// TIA Portal V15.1 export
// export: Created 2024-06-21T08:40:58.6119821Z, ExportSetting WithDefaults, DisplayName Totally Integrated Automation Portal, DisplayVersion V15.1 Update 5, DisplayName TIA Portal Openness, DisplayVersion V15.1 Update 5, DisplayName SINAMICS Startdrive Advanced, DisplayVersion V15.1, DisplayName G130, G150, S120, S150, SINAMICS MV, S210, DisplayVersion V15.1, DisplayName G110M, G120, G120C, G120D, G120P, DisplayVersion V15.1, DisplayName STEP 7 Professional, DisplayVersion V15.1 Update 5, DisplayName STEP 7 Safety, DisplayVersion V15.1, DisplayName WinCC Professional, DisplayVersion V15.1 Update 5, DisplayName SIMATIC Visualization Architect, DisplayVersion V15.1
FUNCTION_BLOCK "LDP/PNCouplerDiag"   // FB1901, FBD
TITLE = LDPCouplerDiag
{ S7_Optimized_Access := 'FALSE' }
AUTHOR : VCC
FAMILY : Communic
NAME : LDPDiag
VERSION : 0.1
// ================================================================================
// Function used to read the diagnostic information from a DP/DP coupler.
// ================================================================================
// stored: AutoNumber false, IsIECCheckEnabled false, SetENOAutomatically False, UDAEnableTagReadback false
   VAR_INPUT
      I_PNPNSendError { ExternalAccessible := 'False'; ExternalVisible := 'False'; ExternalWritable := 'False'} : Bool;   // Send Error
      I_PNPNSendSUBSOn { ExternalAccessible := 'False'; ExternalVisible := 'False'; ExternalWritable := 'False'} : Bool;   // SUBS ON
      I_PNPNDiagSend { ExternalAccessible := 'False'; ExternalVisible := 'False'; ExternalWritable := 'False'} : Byte;   // Diag
      I_PNPNRcvError { ExternalAccessible := 'False'; ExternalVisible := 'False'; ExternalWritable := 'False'} : Bool;   // Recv Error
      I_PNPNRcvSUBSOn { ExternalAccessible := 'False'; ExternalVisible := 'False'; ExternalWritable := 'False'} : Bool;   // SUBS ON
      I_PNPNRcvAckReq { ExternalAccessible := 'False'; ExternalVisible := 'False'; ExternalWritable := 'False'} : Bool;   // ACK REQ
      I_PNPNDiagRecv { ExternalAccessible := 'False'; ExternalVisible := 'False'; ExternalWritable := 'False'} : Byte;   // Diag
      I_AlarmResetPB { ExternalAccessible := 'False'; ExternalVisible := 'False'; ExternalWritable := 'False'} : Bool;   // Alarm reset pushbutton is activated
   END_VAR
   VAR_OUTPUT
      O_Alarm { ExternalAccessible := 'False'; ExternalVisible := 'False'; ExternalWritable := 'False'} : Bool;   // Alarm
      O_AlarmABCondition { ExternalAccessible := 'False'; ExternalVisible := 'False'; ExternalWritable := 'False'} : Bool;   // Alarms AB condition
      H_IAnim { ExternalAccessible := 'False'; ExternalVisible := 'False'; ExternalWritable := 'False'} : Word;   // Icon Animation
   END_VAR
   VAR DB_SPECIFIC
      H_Out : Struct   // HMI
         Anim : Word;   // HMI Animation of the object
         DBnr : Int;   // HMI Animation DB number
      END_STRUCT;
      Alarm { ExternalAccessible := 'False'; ExternalVisible := 'False'; ExternalWritable := 'False'} : Bool;   // Alarm
      Send_error { ExternalAccessible := 'False'; ExternalVisible := 'False'; ExternalWritable := 'False'} : Bool;   // Send Error
      Send_SubOn { ExternalAccessible := 'False'; ExternalVisible := 'False'; ExternalWritable := 'False'} : Bool;   // Send sub on
      Send_TimeOut { ExternalAccessible := 'False'; ExternalVisible := 'False'; ExternalWritable := 'False'} : Bool;   // Send time out
      Send_SeqNrError { ExternalAccessible := 'False'; ExternalVisible := 'False'; ExternalWritable := 'False'} : Bool;   // Send sequenz number error
      Send_CRCError { ExternalAccessible := 'False'; ExternalVisible := 'False'; ExternalWritable := 'False'} : Bool;   // Send CRC error
      Receive_Error { ExternalAccessible := 'False'; ExternalVisible := 'False'; ExternalWritable := 'False'} : Bool;   // Receive error
      Receive_SubOn { ExternalAccessible := 'False'; ExternalVisible := 'False'; ExternalWritable := 'False'} : Bool;   // Receive sub on
      Receive_AckReq { ExternalAccessible := 'False'; ExternalVisible := 'False'; ExternalWritable := 'False'} : Bool;   // Reveice ack request
      Receive_TimeOut { ExternalAccessible := 'False'; ExternalVisible := 'False'; ExternalWritable := 'False'} : Bool;   // Receive time out
      Receive_SeqNrError { ExternalAccessible := 'False'; ExternalVisible := 'False'; ExternalWritable := 'False'} : Bool;   // Receive sequenz number error
      Receive_CRCError { ExternalAccessible := 'False'; ExternalVisible := 'False'; ExternalWritable := 'False'} : Bool;   // Receive CRC error
      AlarmCond { ExternalAccessible := 'False'; ExternalVisible := 'False'; ExternalWritable := 'False'} : Bool;   // Alarm condition
      DBnr { ExternalAccessible := 'False'; ExternalVisible := 'False'; ExternalWritable := 'False'} : Int;   // HMI DB number
   END_VAR
BEGIN

NETWORK
TITLE = **** 1 - Inputs **** DB number
// DB number
      L     DINO;
      T     #DBnr;

REGION Network 2: **** 1 - Inputs **** Information SEND
   // Information SEND
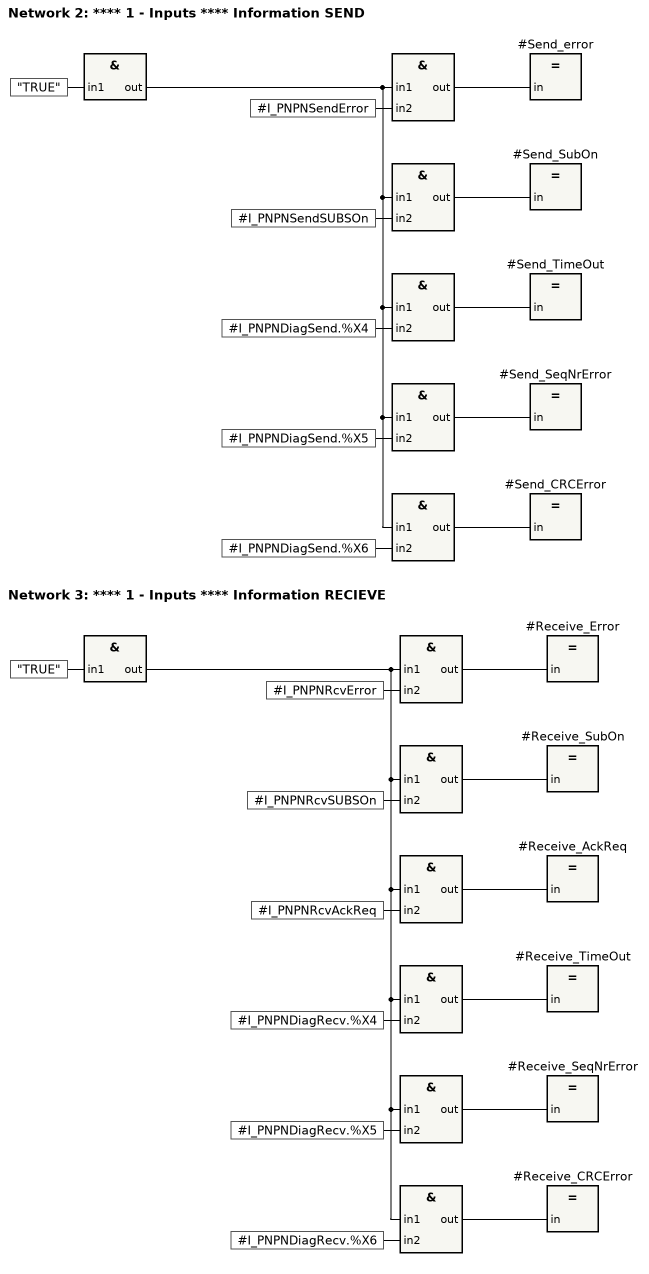
   #Send_error := "TRUE" AND #I_PNPNSendError;
   #Send_SubOn := "TRUE" AND #I_PNPNSendSUBSOn;
   #Send_TimeOut := "TRUE" AND #I_PNPNDiagSend.%X4;
   #Send_SeqNrError := "TRUE" AND #I_PNPNDiagSend.%X5;
   #Send_CRCError := "TRUE" AND #I_PNPNDiagSend.%X6;
END_REGION

REGION Network 3: **** 1 - Inputs **** Information RECIEVE
   // Information RECIEVE
   #Receive_Error := "TRUE" AND #I_PNPNRcvError;
   #Receive_SubOn := "TRUE" AND #I_PNPNRcvSUBSOn;
   #Receive_AckReq := "TRUE" AND #I_PNPNRcvAckReq;
   #Receive_TimeOut := "TRUE" AND #I_PNPNDiagRecv.%X4;
   #Receive_SeqNrError := "TRUE" AND #I_PNPNDiagRecv.%X5;
   #Receive_CRCError := "TRUE" AND #I_PNPNDiagRecv.%X6;
END_REGION

REGION Network 4: **** 2.2 - Alarms - Alarm generation **** Condition send/Recive alarm
   // Condition send/Recive alarm
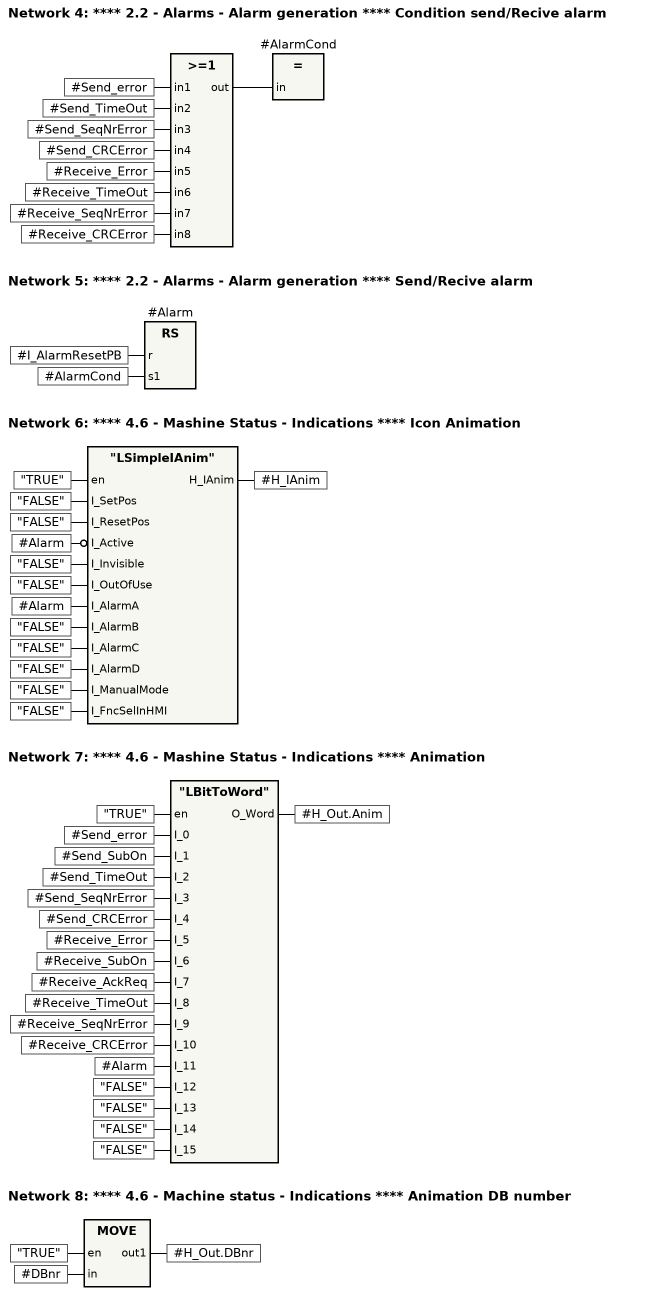
   #AlarmCond := #Send_error OR #Send_TimeOut OR #Send_SeqNrError OR #Send_CRCError OR #Receive_Error OR #Receive_TimeOut OR #Receive_SeqNrError OR #Receive_CRCError;
END_REGION

REGION Network 5: **** 2.2 - Alarms - Alarm generation **** Send/Recive alarm
   // Send/Recive alarm
   IF #I_AlarmResetPB THEN
       #Alarm := FALSE;   // RS flip-flop
   END_IF;
   IF #AlarmCond THEN #Alarm := TRUE; END_IF;
END_REGION

REGION Network 6: **** 4.6 - Mashine Status - Indications **** Icon Animation
   // Icon Animation
   IF "TRUE" THEN
       "LSimpleIAnim"(I_SetPos := "FALSE",
                      I_ResetPos := "FALSE",
                      I_Active := NOT #Alarm,
                      I_Invisible := "FALSE",
                      I_OutOfUse := "FALSE",
                      I_AlarmA := #Alarm,
                      I_AlarmB := "FALSE",
                      I_AlarmC := "FALSE",
                      I_AlarmD := "FALSE",
                      I_ManualMode := "FALSE",
                      I_FncSelInHMI := "FALSE",
                      H_IAnim => #H_IAnim);
   END_IF;
END_REGION

REGION Network 7: **** 4.6 - Mashine Status - Indications **** Animation
   // Animation
   IF "TRUE" THEN
       "LBitToWord"(I_0 := #Send_error,
                    I_1 := #Send_SubOn,
                    I_2 := #Send_TimeOut,
                    I_3 := #Send_SeqNrError,
                    I_4 := #Send_CRCError,
                    I_5 := #Receive_Error,
                    I_6 := #Receive_SubOn,
                    I_7 := #Receive_AckReq,
                    I_8 := #Receive_TimeOut,
                    I_9 := #Receive_SeqNrError,
                    I_10 := #Receive_CRCError,
                    I_11 := #Alarm,
                    I_12 := "FALSE",
                    I_13 := "FALSE",
                    I_14 := "FALSE",
                    I_15 := "FALSE",
                    O_Word => #H_Out.Anim);
   END_IF;
END_REGION

REGION Network 8: **** 4.6 - Machine status - Indications **** Animation DB number
   // Animation DB number
   IF "TRUE" THEN #H_Out.DBnr := #DBnr; END_IF;
END_REGION

REGION Network 9: **** 8 - Outputs **** Alarm
   // Alarm
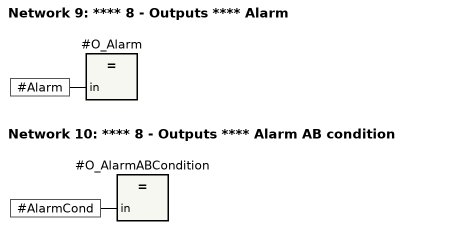
   #O_Alarm := #Alarm;
END_REGION

REGION Network 10: **** 8 - Outputs **** Alarm AB condition
   // Alarm AB condition
   #O_AlarmABCondition := #AlarmCond;
END_REGION
END_FUNCTION_BLOCK
